SYSTEM Teste_01
  (* Version 1.0, 2025-02-03, FESTO *)
  APPLICATION Teste_01App
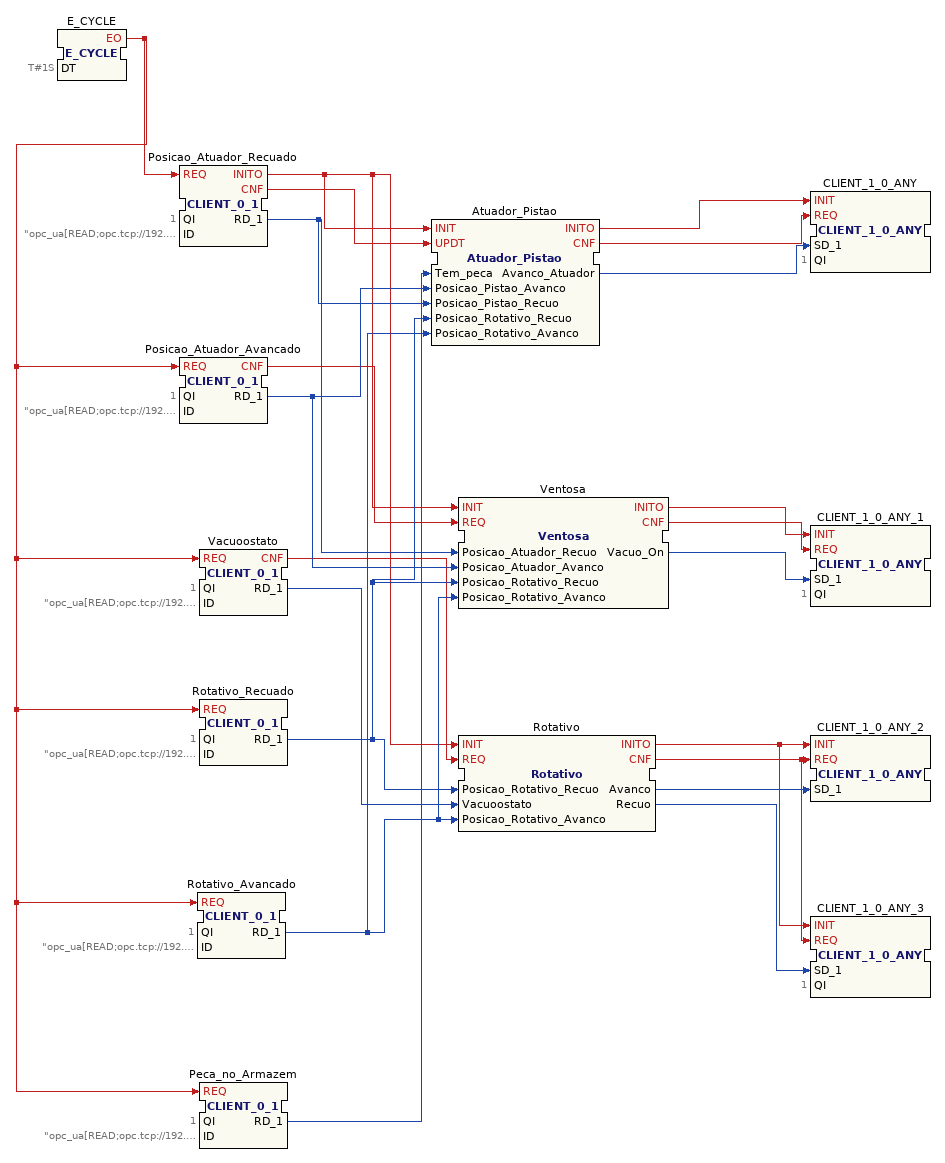
    FBS
      Posicao_Atuador_Recuado : CLIENT_0_1(QI := 1, ID := "opc_ua[READ;opc.tcp://192.168.2.20:4840#;,2:s=|var|CPX-CEC-C1-V3.Application.PLC_PRG.posicao_atuador_avancoo]");
      E_CYCLE : E_CYCLE(DT := T#1S);
      Posicao_Atuador_Avancado : CLIENT_0_1(QI := 1, ID := "opc_ua[READ;opc.tcp://192.168.2.20:4840#;,2:s=|var|CPX-CEC-C1-V3.Application.PLC_PRG.posicao_atuador_recuoo]");
      Vacuoostato : CLIENT_0_1(QI := 1, ID := "opc_ua[READ;opc.tcp://192.168.2.20:4840#;,2:s=|var|CPX-CEC-C1-V3.Application.PLC_PRG.vacuostatoo]"); (* Se tem peca ou não na ventosa *)
      Rotativo_Recuado : CLIENT_0_1(QI := 1, ID := "opc_ua[READ;opc.tcp://192.168.2.20:4840#;,2:s=|var|CPX-CEC-C1-V3.Application.PLC_PRG.posicao_rotativo_recuoo]");
      Rotativo_Avancado : CLIENT_0_1(QI := 1, ID := "opc_ua[READ;opc.tcp://192.168.2.20:4840#;,2:s=|var|CPX-CEC-C1-V3.Application.PLC_PRG.posicao_rotativo_avancoo]");
      Peca_no_Armazem : CLIENT_0_1(QI := 1, ID := "opc_ua[READ;opc.tcp://192.168.2.20:4840#;,2:s=|var|CPX-CEC-C1-V3.Application.PLC_PRG.peca_aramzemm]");
      Atuador_Pistao : Atuador_Pistao;
      Rotativo : Rotativo;
      Ventosa : Ventosa;
      CLIENT_1_0_ANY : CLIENT_1_0_ANY(QI := 1);
      CLIENT_1_0_ANY_1 : CLIENT_1_0_ANY(QI := 1);
      CLIENT_1_0_ANY_2 : CLIENT_1_0_ANY;
      CLIENT_1_0_ANY_3 : CLIENT_1_0_ANY(QI := 1);
    END_FBS
    EVENT_CONNECTIONS
      E_CYCLE.EO TO Posicao_Atuador_Recuado.REQ;
      E_CYCLE.EO TO Posicao_Atuador_Avancado.REQ;
      E_CYCLE.EO TO Vacuoostato.REQ;
      E_CYCLE.EO TO Rotativo_Recuado.REQ;
      E_CYCLE.EO TO Rotativo_Avancado.REQ;
      E_CYCLE.EO TO Peca_no_Armazem.REQ;
      Posicao_Atuador_Recuado.INITO TO Atuador_Pistao.INIT;
      Posicao_Atuador_Recuado.INITO TO Ventosa.INIT;
      Posicao_Atuador_Recuado.INITO TO Rotativo.INIT;
      Posicao_Atuador_Recuado.CNF TO Atuador_Pistao.UPDT;
      Posicao_Atuador_Avancado.CNF TO Ventosa.REQ;
      Vacuoostato.CNF TO Rotativo.REQ;
      Atuador_Pistao.INITO TO CLIENT_1_0_ANY.INIT;
      Atuador_Pistao.CNF TO CLIENT_1_0_ANY.REQ;
      Ventosa.INITO TO CLIENT_1_0_ANY_1.INIT;
      Ventosa.CNF TO CLIENT_1_0_ANY_1.REQ;
      Rotativo.INITO TO CLIENT_1_0_ANY_2.INIT;
      Rotativo.CNF TO CLIENT_1_0_ANY_2.REQ;
      Rotativo.INITO TO CLIENT_1_0_ANY_3.INIT;
      Rotativo.CNF TO CLIENT_1_0_ANY_3.REQ;
    END_CONNECTIONS
    DATA_CONNECTIONS
      Peca_no_Armazem.RD_1 TO Atuador_Pistao.Tem_peca;
      Posicao_Atuador_Avancado.RD_1 TO Atuador_Pistao.Posicao_Pistao_Avanco;
      Posicao_Atuador_Recuado.RD_1 TO Atuador_Pistao.Posicao_Pistao_Recuo;
      Rotativo_Recuado.RD_1 TO Atuador_Pistao.Posicao_Rotativo_Recuo;
      Rotativo_Avancado.RD_1 TO Atuador_Pistao.Posicao_Rotativo_Avanco;
      Posicao_Atuador_Recuado.RD_1 TO Ventosa.Posicao_Atuador_Recuo;
      Posicao_Atuador_Avancado.RD_1 TO Ventosa.Posicao_Atuador_Avanco;
      Rotativo_Recuado.RD_1 TO Ventosa.Posicao_Rotativo_Recuo;
      Rotativo_Avancado.RD_1 TO Ventosa.Posicao_Rotativo_Avanco;
      Rotativo_Recuado.RD_1 TO Rotativo.Posicao_Rotativo_Recuo;
      Vacuoostato.RD_1 TO Rotativo.Vacuoostato;
      Rotativo_Avancado.RD_1 TO Rotativo.Posicao_Rotativo_Avanco;
      Atuador_Pistao.Avanco_Atuador TO CLIENT_1_0_ANY.SD_1;
      Ventosa.Vacuo_On TO CLIENT_1_0_ANY_1.SD_1;
      Rotativo.Avanco TO CLIENT_1_0_ANY_2.SD_1;
      Rotativo.Recuo TO CLIENT_1_0_ANY_3.SD_1;
    END_CONNECTIONS
  END_APPLICATION
  DEVICE FORTE_PC : FORTE_PC(MGR_ID := "localhost:61499")
    {SET_ATTRIBUTE(Profile, HOLOBLOC)} (* device profile *)
    RESOURCE EMB_RES : EMB_RES
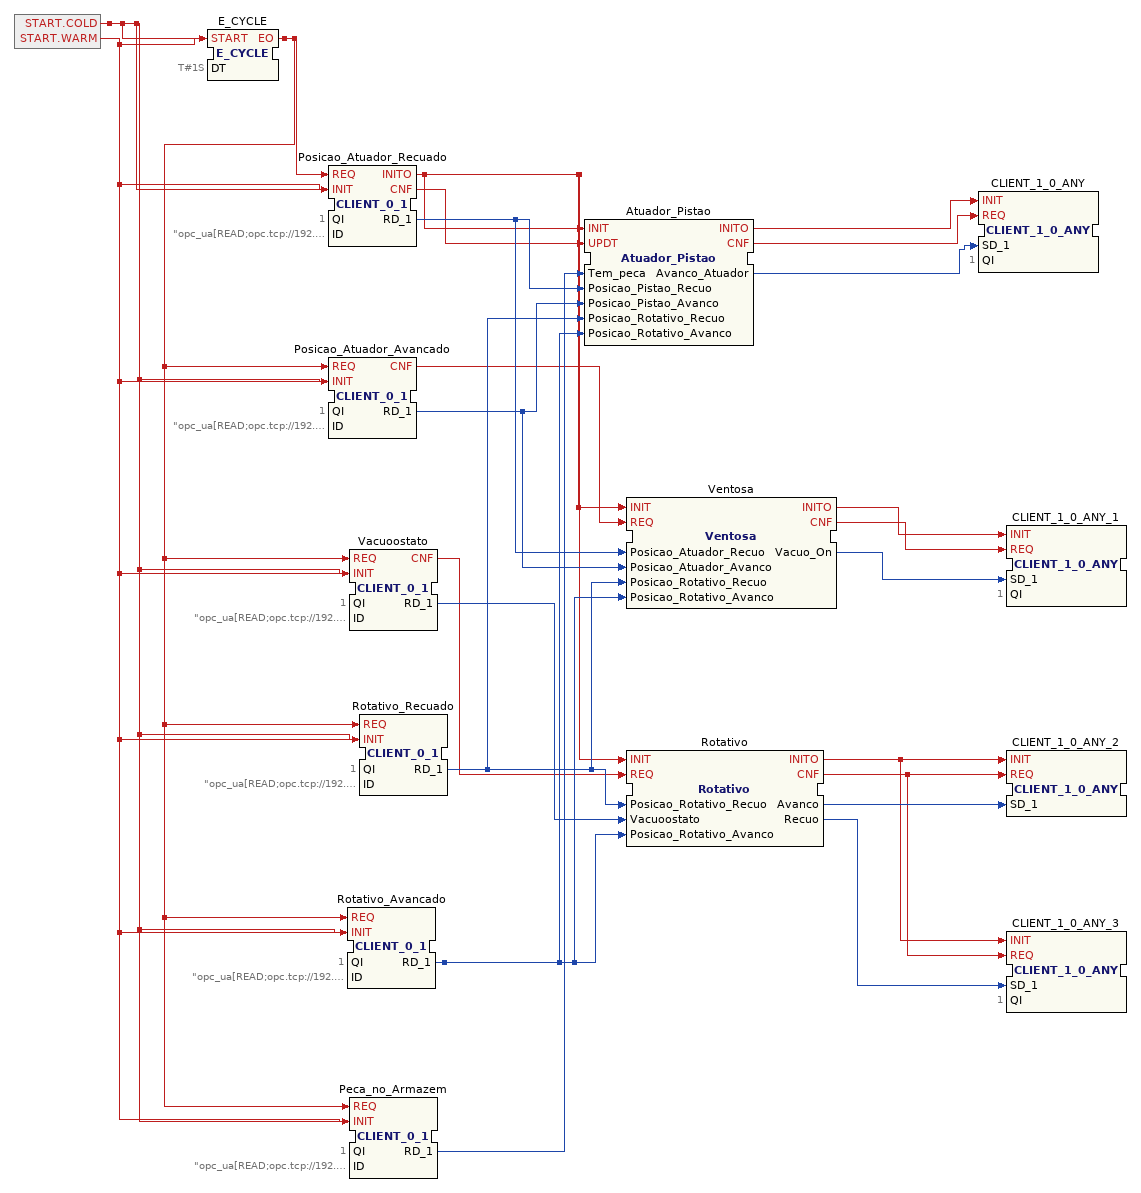
      FBS
        Posicao_Atuador_Recuado : CLIENT_0_1(QI := 1, ID := "opc_ua[READ;opc.tcp://192.168.2.20:4840#;,2:s=|var|CPX-CEC-C1-V3.Application.PLC_PRG.posicao_atuador_avancoo]");
        E_CYCLE : E_CYCLE(DT := T#1S);
        Posicao_Atuador_Avancado : CLIENT_0_1(QI := 1, ID := "opc_ua[READ;opc.tcp://192.168.2.20:4840#;,2:s=|var|CPX-CEC-C1-V3.Application.PLC_PRG.posicao_atuador_recuoo]");
        Vacuoostato : CLIENT_0_1(QI := 1, ID := "opc_ua[READ;opc.tcp://192.168.2.20:4840#;,2:s=|var|CPX-CEC-C1-V3.Application.PLC_PRG.vacuostatoo]");
        Rotativo_Recuado : CLIENT_0_1(QI := 1, ID := "opc_ua[READ;opc.tcp://192.168.2.20:4840#;,2:s=|var|CPX-CEC-C1-V3.Application.PLC_PRG.posicao_rotativo_recuoo]");
        Rotativo_Avancado : CLIENT_0_1(QI := 1, ID := "opc_ua[READ;opc.tcp://192.168.2.20:4840#;,2:s=|var|CPX-CEC-C1-V3.Application.PLC_PRG.posicao_rotativo_avancoo]");
        Peca_no_Armazem : CLIENT_0_1(QI := 1, ID := "opc_ua[READ;opc.tcp://192.168.2.20:4840#;,2:s=|var|CPX-CEC-C1-V3.Application.PLC_PRG.peca_aramzemm]");
        Atuador_Pistao : Atuador_Pistao;
        Ventosa : Ventosa;
        Rotativo : Rotativo;
        CLIENT_1_0_ANY : CLIENT_1_0_ANY(QI := 1);
        CLIENT_1_0_ANY_1 : CLIENT_1_0_ANY(QI := 1);
        CLIENT_1_0_ANY_2 : CLIENT_1_0_ANY;
        CLIENT_1_0_ANY_3 : CLIENT_1_0_ANY(QI := 1);
      END_FBS
      EVENT_CONNECTIONS
        E_CYCLE.EO TO Posicao_Atuador_Recuado.REQ;
        START.COLD TO E_CYCLE.START;
        START.WARM TO E_CYCLE.START;
        START.COLD TO Posicao_Atuador_Recuado.INIT;
        START.WARM TO Posicao_Atuador_Recuado.INIT;
        E_CYCLE.EO TO Posicao_Atuador_Avancado.REQ;
        E_CYCLE.EO TO Vacuoostato.REQ;
        E_CYCLE.EO TO Rotativo_Recuado.REQ;
        E_CYCLE.EO TO Rotativo_Avancado.REQ;
        E_CYCLE.EO TO Peca_no_Armazem.REQ;
        START.WARM TO Posicao_Atuador_Avancado.INIT;
        START.COLD TO Posicao_Atuador_Avancado.INIT;
        START.WARM TO Vacuoostato.INIT;
        START.COLD TO Vacuoostato.INIT;
        START.WARM TO Rotativo_Recuado.INIT;
        START.COLD TO Rotativo_Recuado.INIT;
        START.WARM TO Rotativo_Avancado.INIT;
        START.COLD TO Rotativo_Avancado.INIT;
        START.COLD TO Peca_no_Armazem.INIT;
        START.WARM TO Peca_no_Armazem.INIT;
        Posicao_Atuador_Recuado.INITO TO Atuador_Pistao.INIT;
        Posicao_Atuador_Recuado.INITO TO Ventosa.INIT;
        Posicao_Atuador_Recuado.INITO TO Rotativo.INIT;
        Posicao_Atuador_Recuado.CNF TO Atuador_Pistao.UPDT;
        Posicao_Atuador_Avancado.CNF TO Ventosa.REQ;
        Vacuoostato.CNF TO Rotativo.REQ;
        Atuador_Pistao.INITO TO CLIENT_1_0_ANY.INIT;
        Atuador_Pistao.CNF TO CLIENT_1_0_ANY.REQ;
        Ventosa.INITO TO CLIENT_1_0_ANY_1.INIT;
        Ventosa.CNF TO CLIENT_1_0_ANY_1.REQ;
        Rotativo.INITO TO CLIENT_1_0_ANY_2.INIT;
        Rotativo.CNF TO CLIENT_1_0_ANY_2.REQ;
        Rotativo.INITO TO CLIENT_1_0_ANY_3.INIT;
        Rotativo.CNF TO CLIENT_1_0_ANY_3.REQ;
      END_CONNECTIONS
      DATA_CONNECTIONS
        Peca_no_Armazem.RD_1 TO Atuador_Pistao.Tem_peca;
        Posicao_Atuador_Recuado.RD_1 TO Atuador_Pistao.Posicao_Pistao_Recuo;
        Posicao_Atuador_Avancado.RD_1 TO Atuador_Pistao.Posicao_Pistao_Avanco;
        Rotativo_Recuado.RD_1 TO Atuador_Pistao.Posicao_Rotativo_Recuo;
        Rotativo_Avancado.RD_1 TO Atuador_Pistao.Posicao_Rotativo_Avanco;
        Posicao_Atuador_Recuado.RD_1 TO Ventosa.Posicao_Atuador_Recuo;
        Posicao_Atuador_Avancado.RD_1 TO Ventosa.Posicao_Atuador_Avanco;
        Rotativo_Recuado.RD_1 TO Ventosa.Posicao_Rotativo_Recuo;
        Rotativo_Avancado.RD_1 TO Ventosa.Posicao_Rotativo_Avanco;
        Rotativo_Recuado.RD_1 TO Rotativo.Posicao_Rotativo_Recuo;
        Vacuoostato.RD_1 TO Rotativo.Vacuoostato;
        Rotativo_Avancado.RD_1 TO Rotativo.Posicao_Rotativo_Avanco;
        Atuador_Pistao.Avanco_Atuador TO CLIENT_1_0_ANY.SD_1;
        Ventosa.Vacuo_On TO CLIENT_1_0_ANY_1.SD_1;
        Rotativo.Avanco TO CLIENT_1_0_ANY_2.SD_1;
        Rotativo.Recuo TO CLIENT_1_0_ANY_3.SD_1;
      END_CONNECTIONS
    END_RESOURCE
  END_DEVICE
  MAPPINGS
    Teste_01App.Posicao_Atuador_Recuado ON FORTE_PC.EMB_RES.Posicao_Atuador_Recuado;
    Teste_01App.E_CYCLE ON FORTE_PC.EMB_RES.E_CYCLE;
    Teste_01App.Posicao_Atuador_Avancado ON FORTE_PC.EMB_RES.Posicao_Atuador_Avancado;
    Teste_01App.Vacuoostato ON FORTE_PC.EMB_RES.Vacuoostato;
    Teste_01App.Rotativo_Recuado ON FORTE_PC.EMB_RES.Rotativo_Recuado;
    Teste_01App.Rotativo_Avancado ON FORTE_PC.EMB_RES.Rotativo_Avancado;
    Teste_01App.Peca_no_Armazem ON FORTE_PC.EMB_RES.Peca_no_Armazem;
    Teste_01App.Atuador_Pistao ON FORTE_PC.EMB_RES.Atuador_Pistao;
    Teste_01App.Ventosa ON FORTE_PC.EMB_RES.Ventosa;
    Teste_01App.Rotativo ON FORTE_PC.EMB_RES.Rotativo;
    Teste_01App.CLIENT_1_0_ANY ON FORTE_PC.EMB_RES.CLIENT_1_0_ANY;
    Teste_01App.CLIENT_1_0_ANY_1 ON FORTE_PC.EMB_RES.CLIENT_1_0_ANY_1;
    Teste_01App.CLIENT_1_0_ANY_2 ON FORTE_PC.EMB_RES.CLIENT_1_0_ANY_2;
    Teste_01App.CLIENT_1_0_ANY_3 ON FORTE_PC.EMB_RES.CLIENT_1_0_ANY_3;
  END_MAPPINGS
  SEGMENTS
    Ethernet : Ethernet;
  END_SEGMENTS
  LINKS
    FORTE_PC => Ethernet;
  END_LINKS
END_SYSTEM
